(* IEC 61131-3 sources: jiepp/tests/jiepp/input/D_option, 1 file *)

(* ---- D_option.iec ---- *)
program POU
var
    v: int := INITIAL_VALUE;
end_var

v := EXPR;

end_program
